PROGRAM myCNC_Call_Place
VAR
END_VAR

END_PROGRAM

(* stored: Version 1.1.0.1, ProductVersion 3.1.4024.11
   POU myCNC_Call_Place: Id {54d01624-1da8-4928-847e-78947d3f846d}, SpecialFunc None *)
